// Mitsubishi GX Works2 project: 230930-001- exercicios-0-1   PLC: Q03UDV

// task Task_01 (event TRUE, interval 0, priority 31): POU_01

PROGRAM POU_01
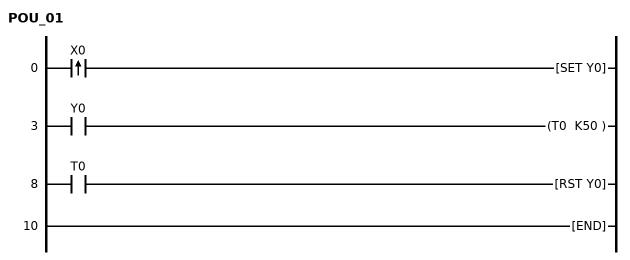
0     LDP     X0
      SET     Y0
3     LD      Y0
      OUT     T0 K50
8     LD      T0
      RST     Y0
10    END
END_PROGRAM
